FUNCTION_BLOCK PUSHER_CTRL (* Composite Function Block Type *)
  (* Standard: 61499-2 *)
  (* Version 0.2, 2003-12-05, JHC, Rockwell Automation, Renamed from NEWCOMPFB. *)
  (* Version 0.1, 2002-01-08, JHC, Rockwell Automation, Added DLY FB as example. *)
  (* Version 0.0, 2000-05-27, JHC, Rockwell Automation *)
  (* Compiler header: package fb.rt.dasdA1.A2; *)
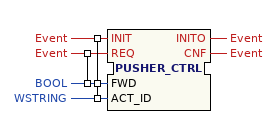
  EVENT_INPUT
    INIT WITH FWD, ACT_ID; (* Initialization Request *)
    REQ WITH FWD; (* Normal Execution Request *)
  END_EVENT
  EVENT_OUTPUT
    INITO; (* Initialization Confirm *)
    CNF; (* Execution Confirmation *)
  END_EVENT
  VAR_INPUT
    FWD : BOOL; (* Input event qualifier *)
    ACT_ID : WSTRING;
  END_VAR
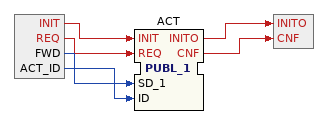
  FBS
    ACT : PUBL_1;
  END_FBS
  EVENT_CONNECTIONS
    INIT TO ACT.INIT;
    ACT.INITO TO INITO;
    REQ TO ACT.REQ;
    ACT.CNF TO CNF;
  END_CONNECTIONS
  DATA_CONNECTIONS
    FWD TO ACT.SD_1;
    ACT_ID TO ACT.ID;
  END_CONNECTIONS
END_FUNCTION_BLOCK
